(* CODESYS project building automation.project

Project tree, tasks and I/O mapping:
  Device : L-force Controller c300 Logic, Lenze, order no. LPC 1000, version 3.8.0.0
    application Application
      libraries: L_Util, 3.3.0.0 (Lenze); L_PLCDataManagerAccess, 3.0.0.0 (Lenze); L_PLCLoggingAccess, 3.3.0.0 (Lenze)
      task MainTask (cyclic, interval t#10ms, priority 1) calls PLC_PRG
      program PLC_PRG [LD]
    Coupler_I_O_moduls : Coupler I/O moduls, Lenze, version 3.6.0.0
        settings: Count groups = 1; Application Name of Task = 'Application'; Group1 Task Name = 'MainTask'
        unmapped channels: Error, unused, unused, unused, unused, unused, unused, unused, ErrorID, AbsoluteCounter, ErrorReset, unused, unused, unused, unused, unused, unused, unused
      EPM_S202 : EPM-S202: DI8, DC 24V, Lenze, order no. EPM-S202, version 3.6.0.0
          settings: Group = 0; Task Guid = '00000000-0000-0000-0000-000000000000'
          input  Application.PLC_PRG.xDoorStateLocked : BIT  // DI1
          input  Application.PLC_PRG.xdoorStateUnlocked : BIT  // DI2
          input  Application.PLC_PRG.xMasterAlarmReset : BIT  // DI3
          input  Application.PLC_PRG.xEndofDayInput : BIT  // DI4
          input  Application.PLC_PRG.xStartofDayInput : BIT  // DI5
          input  Application.PLC_PRG.xDoor_1_Open : BIT  // DI6
          input  Application.PLC_PRG.xDoorCodeInput : BIT  // DI7
          input  Application.PLC_PRG.xInteriorDoorSensor : BIT  // DI8
      EPM_S302 : EPM-S302: DO8, DC 24V, 0.5A, Lenze, order no. EPM-S302, version 3.6.0.0
          settings: Group = 0; Task Guid = '00000000-0000-0000-0000-000000000000'
          output Application.PLC_PRG.xDoor_1_Lock : BIT  // DO1
          output Application.PLC_PRG.xfireAlarm : BIT  // DO2
          output Application.PLC_PRG.xset_EndofDay : BIT  // DO3
          output Application.PLC_PRG.xSet_falseEntryAlarm : BIT  // DO4
          output Application.PLC_PRG.xset_doorUnlockedbyCode : BIT  // DO5
          output Application.PLC_PRG.xDoor_1_Open : BIT  // DO6
          unmapped channels: DO7, DO8
      EPM_S202_1 : EPM-S202: DI8, DC 24V, Lenze, order no. EPM-S202, version 3.6.0.0
          settings: Group = 0; Task Guid = '00000000-0000-0000-0000-000000000000'
          input  Application.PLC_PRG.xfireAlarmInput : BIT  // DI1
          unmapped channels: DI2, DI3, DI4, DI5, DI6, DI7, DI8
*)

// Device/Application/PLC_PRG
PROGRAM PLC_PRG

VAR
	xDoorStateLocked: BOOL;
	xset_doorStateLocked: BOOL;
	xDoor_1_Lock: BOOL;
	xset_doorStateUnlocked: BOOL;
	xdoorStateUnlocked: BOOL;
	xfireAlarm: BOOL;
	xset_fireAlarm: BOOL;
	xMasterAlarmReset: BOOL;
	xset_masterAlarmReset: BOOL;
	xEndofDayInput: BOOL;
	xroom216MotionSensor: BOOL;
	xset_EndofDay: BOOL;
	xSet_falseEntryAlarm: BOOL;
	xDoor_1_Open: BOOL;
	xset_EndofDayInput: BOOL;
	xStartofDayInput: BOOL;
	xset_StartofdayInput: BOOL;
	xDoorCodeInput: BOOL;
	xset_DoorCodeUnlocked: BOOL;
	xset_doorUnlockedbyCode: BOOL;
	xset_doorCodeLocked: BOOL;
	xcodeUnlockedCondition: BOOL;
	xDoorCodeInputLatch: BOOL;
	delay1: TON;
	delay2: TON;
	delay3: TON;
	xInteriorDoorSensor: BOOL;
	delay4: TON;
	xfireAlarmInput: BOOL;
END_VAR
VAR // added by the converter: edge detectors and wires of the graphical bodies
    _w1, _w2, _w3, _w4, _w5, _w6, _w7 : BOOL;
END_VAR

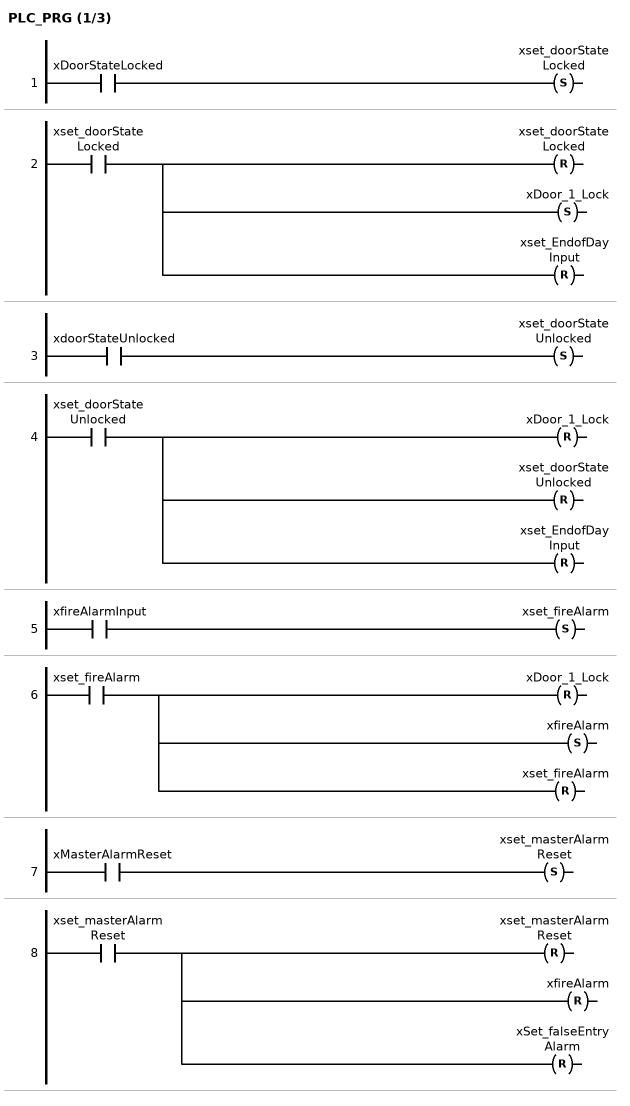
// NETWORK 1
xset_doorStateLocked S= xDoorStateLocked;

// NETWORK 2
_w1 := xset_doorStateLocked;
xset_doorStateLocked R= _w1;
xDoor_1_Lock S= _w1;
xset_EndofDayInput R= _w1;

// NETWORK 3
xset_doorStateUnlocked S= xdoorStateUnlocked;

// NETWORK 4
_w2 := xset_doorStateUnlocked;
xDoor_1_Lock R= _w2;
xset_doorStateUnlocked R= _w2;
xset_EndofDayInput R= _w2;

// NETWORK 5
xset_fireAlarm S= xfireAlarmInput;

// NETWORK 6
xDoor_1_Lock R= xset_fireAlarm;
xfireAlarm S= xset_fireAlarm;
xset_fireAlarm R= xset_fireAlarm;

// NETWORK 7
xset_masterAlarmReset S= xMasterAlarmReset;

// NETWORK 8
_w3 := xset_masterAlarmReset;
xset_masterAlarmReset R= _w3;
xfireAlarm R= _w3;
xSet_falseEntryAlarm R= _w3;

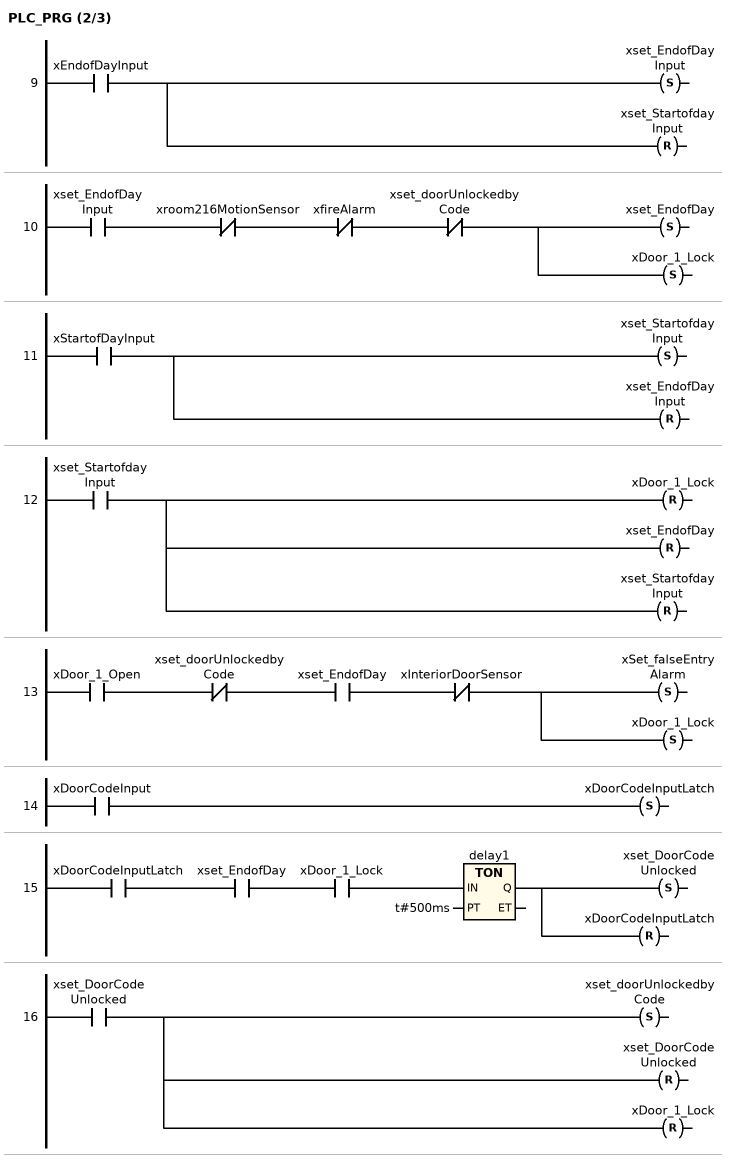
// NETWORK 9
xset_EndofDayInput S= xEndofDayInput;
xset_StartofdayInput R= xEndofDayInput;

// NETWORK 10
_w4 := xset_EndofDayInput AND NOT xroom216MotionSensor AND NOT xfireAlarm AND NOT xset_doorUnlockedbyCode;
xset_EndofDay S= _w4;
xDoor_1_Lock S= _w4;

// NETWORK 11
xset_StartofdayInput S= xStartofDayInput;
xset_EndofDayInput R= xStartofDayInput;

// NETWORK 12
xDoor_1_Lock R= xset_StartofdayInput;
xset_EndofDay R= xset_StartofdayInput;
xset_StartofdayInput R= xset_StartofdayInput;

// NETWORK 13
_w5 := xDoor_1_Open AND NOT xset_doorUnlockedbyCode AND xset_EndofDay AND NOT xInteriorDoorSensor;
xSet_falseEntryAlarm S= _w5;
xDoor_1_Lock S= _w5;

// NETWORK 14
xDoorCodeInputLatch S= xDoorCodeInput;

// NETWORK 15
delay1(IN := xDoorCodeInputLatch AND xset_EndofDay AND xDoor_1_Lock, PT := t#500ms); // TON
xset_DoorCodeUnlocked S= delay1.Q;
xDoorCodeInputLatch R= delay1.Q;

// NETWORK 16
_w6 := xset_DoorCodeUnlocked;
xset_doorUnlockedbyCode S= _w6;
xset_DoorCodeUnlocked R= _w6;
xDoor_1_Lock R= _w6;

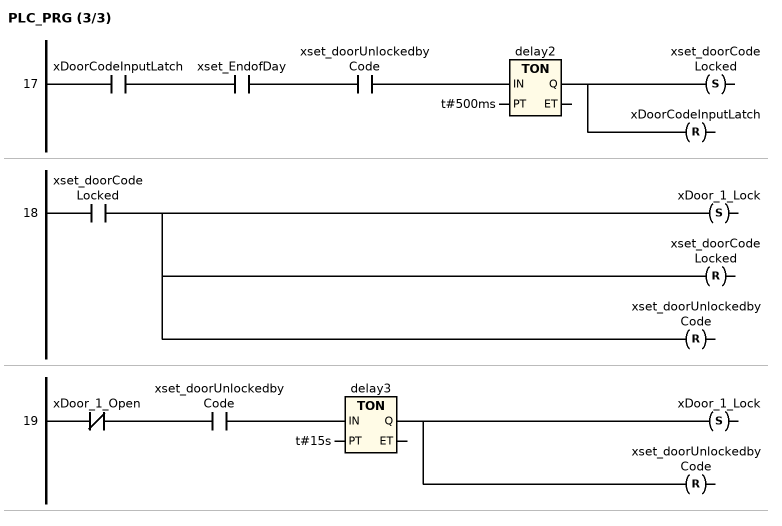
// NETWORK 17
delay2(IN := xDoorCodeInputLatch AND xset_EndofDay AND xset_doorUnlockedbyCode, PT := t#500ms); // TON
xset_doorCodeLocked S= delay2.Q;
xDoorCodeInputLatch R= delay2.Q;

// NETWORK 18
_w7 := xset_doorCodeLocked;
xDoor_1_Lock S= _w7;
xset_doorCodeLocked R= _w7;
xset_doorUnlockedbyCode R= _w7;

// NETWORK 19
delay3(IN := NOT xDoor_1_Open AND xset_doorUnlockedbyCode, PT := t#15s); // TON
xDoor_1_Lock S= delay3.Q;
xset_doorUnlockedbyCode R= delay3.Q;

END_PROGRAM
